Fanuc KAREL source: ko00032.KL

-- PROVISIONAL review KL for V1013-1; original PC SHA256 73368d97e262d5b220221db27a7cb961b4f62396b62126c0867d82568f4e030d
-- Incomplete behavior may be omitted. Consult companion uncertainty JSON. Do not deploy.
PROGRAM KO00032
%NOLOCKGROUP
-- UNRESOLVED_DECL P1 type=000199
-- UNRESOLVED_DECL P2 type=000199
-- UNRESOLVED_DECL P3 type=000199
-- UNRESOLVED_DECL P4 type=000199
-- UNRESOLVED_DECL OUT type=000199
BEGIN
  -- UNRESOLVED_PC offsets 5-80; opcodes 27,27,49,7E,AD,27,49,7E,AD,27,49,7E,AD,27,49,7E,AD,76,7E,4A
  -- UNRESOLVED_PC offsets 85-89; opcodes 7F
END KO00032
